// TwinCAT 3 PLC project State_Pattern
// Title: State Pattern PackML
// Company: ChrisK
// ProjectVersion: 0.0.0.1
// ProgramVersion: 3.1.4023.0
// libraries:
//   Tc2_Standard, * (Beckhoff Automation GmbH)
//   Tc2_System, * (Beckhoff Automation GmbH)
//   Tc3_Module, * (Beckhoff Automation GmbH)
//   Tc3_PackML_V2, * (Beckhoff Automation GmbH)
// project tree:
//   PackML_Method_Pattern/ PML_Method_Base.TcPOU
//   PackML_State_Pattern/ Aborted_State.TcPOU, Aborting_State.TcPOU, Clearing_State.TcPOU, Execute_State.TcPOU, Idle_State.TcPOU, ITF_State.TcIO, PML_StatePattern_Base.TcPOU, Resetting_State.TcPOU, Starting_State.TcPOU, Stopped_State.TcPOU, Undefined_State.TcPOU

// ---- PackML_State_Pattern/ITF_State.TcIO
INTERFACE ITF_State

METHOD Cycle : BOOL
VAR_INPUT
END_VAR
END_METHOD

END_INTERFACE

// ---- PackML_Method_Pattern/PML_Method_Base.TcPOU
FUNCTION_BLOCK PML_Method_Base
VAR_INPUT
END_VAR
VAR_OUTPUT
END_VAR
VAR
	ipackml : IPmlStateMachine;
END_VAR

METHOD PROTECTED Aborted : BOOL
VAR_INPUT
END_VAR
END_METHOD

METHOD PROTECTED Aborting : BOOL
VAR_INPUT
END_VAR
ipackml.SetStateComplete();
END_METHOD

METHOD PROTECTED Clearing : BOOL
VAR_INPUT
END_VAR
ipackml.SetStateComplete();
END_METHOD

METHOD PROTECTED Completed : BOOL
VAR_INPUT
END_VAR
END_METHOD

METHOD PROTECTED Completing : BOOL
VAR_INPUT
END_VAR
ipackml.SetStateComplete();
END_METHOD

METHOD PUBLIC Cycle : BOOL
VAR_INPUT
END_VAR
CASE ipackml.GetCurrentState() OF
	E_PMLState.ePMLState_Clearing:
		Clearing();
	E_PMLState.ePMLState_Aborted:
		Aborted();
	E_PMLState.ePMLState_Aborting:
		Aborting();
	E_PMLState.ePMLState_Complete:
		Completed();
	E_PMLState.ePMLState_Completing:
		Completing();
	E_PMLState.ePMLState_Execute:
		Execute();
	E_PMLState.ePMLState_Held:
		Held();
	E_PMLState.ePMLState_Holding:
		Holding();
	E_PMLState.ePMLState_Idle:
		Idle();
	E_PMLState.ePMLState_Resetting:
		Resetting();
	E_PMLState.ePMLState_Starting:
		Starting();
	E_PMLState.ePMLState_Stopped:
		Stopped();
	E_PMLState.ePMLState_Stopping:
		Stopping();
	E_PMLState.ePMLState_Suspended:
		Suspended();
	E_PMLState.ePMLState_Suspending:
		Suspending();
	E_PMLState.ePMLState_Undefined:
		Undefined();
	E_PMLState.ePMLState_Unholding:
		Unholding();
	E_PMLState.ePMLState_Unsuspending:
		Unsuspending();
END_CASE
END_METHOD

METHOD PROTECTED Execute : BOOL
VAR_INPUT
END_VAR
END_METHOD

METHOD PROTECTED Held : BOOL
VAR_INPUT
END_VAR
END_METHOD

METHOD PROTECTED Holding : BOOL
VAR_INPUT
END_VAR
ipackml.SetStateComplete();
END_METHOD

METHOD PROTECTED Idle : BOOL
VAR_INPUT
END_VAR
END_METHOD

PROPERTY PUBLIC PackMLStateMachine : IPmlStateMachine
GET
PackMLStateMachine := ipackml;
END_GET
SET
ipackml := PackMLStateMachine;
END_SET
END_PROPERTY

METHOD PROTECTED Resetting : BOOL
VAR_INPUT
END_VAR
ipackml.SetStateComplete();
END_METHOD

METHOD PROTECTED Starting : BOOL
VAR_INPUT
END_VAR
ipackml.SetStateComplete();
END_METHOD

METHOD PROTECTED Stopped : BOOL
VAR_INPUT
END_VAR
END_METHOD

METHOD PROTECTED Stopping : BOOL
VAR_INPUT
END_VAR
ipackml.SetStateComplete();
END_METHOD

METHOD PROTECTED Suspended : BOOL
VAR_INPUT
END_VAR
END_METHOD

METHOD PROTECTED Suspending : BOOL
VAR_INPUT
END_VAR
ipackml.SetStateComplete();
END_METHOD

METHOD PROTECTED Undefined : BOOL
VAR_INPUT
END_VAR
END_METHOD

METHOD PROTECTED Unholding : BOOL
VAR_INPUT
END_VAR
ipackml.SetStateComplete();
END_METHOD

METHOD PROTECTED Unsuspending : BOOL
VAR_INPUT
END_VAR
ipackml.SetStateComplete();
END_METHOD

END_FUNCTION_BLOCK

// ---- PackML_State_Pattern/Aborted_State.TcPOU
FUNCTION_BLOCK Aborted_State IMPLEMENTS ITF_State
VAR_INPUT
END_VAR
VAR_OUTPUT
END_VAR
VAR
	pPML_Base : POINTER TO PML_StatePattern_Base;
	_stateMachine : IPmlStateMachine;
END_VAR

METHOD Cycle : BOOL
VAR_INPUT
END_VAR
IF _stateMachine.GetCurrentState() = E_PMLState.ePMLState_Clearing THEN
	pPML_Base^.SetState(pPML_Base^.clearing);
END_IF
END_METHOD

METHOD FB_init : BOOL
VAR_INPUT
	bInitRetains : BOOL; // if TRUE, the retain variables are initialized (warm start / cold start)
	bInCopyCode : BOOL;  // if TRUE, the instance afterwards gets moved into the copy code (online change)
	pPML_Base : POINTER TO PML_StatePattern_Base;
	statemachine : IPmlStateMachine;
END_VAR
_stateMachine := statemachine;
THIS^.pPML_Base := pPML_Base;
END_METHOD

END_FUNCTION_BLOCK

// ---- PackML_State_Pattern/PML_StatePattern_Base.TcPOU
FUNCTION_BLOCK PML_StatePattern_Base
VAR_INPUT
END_VAR
VAR_OUTPUT
END_VAR
VAR
	stateMachine : PMLStateMachine;
	iStateMachine : IPmlStateMachine := stateMachine;
	undefined : Undefined_State(THIS, iStateMachine);
	aborting : Aborting_State(THIS, iStateMachine);
	aborted : Aborted_State(THIS, iStateMachine);
	clearing : Clearing_State(THIS, iStateMachine);
	stopped : Stopped_State(THIS, iStateMachine);
	resetting : Resetting_State(THIS, iStateMachine);
	idle : Idle_State(THIS, iStateMachine);
	starting : Starting_State(THIS, iStateMachine);
	execute : Execute_State(THIS, iStateMachine);
	iState : ITF_State := undefined;
END_VAR

iState.Cycle();
stateMachine();

METHOD SetState : BOOL
VAR_INPUT
  newState : ITF_State;
END_VAR
THIS^.iState := newState;
END_METHOD

END_FUNCTION_BLOCK

// ---- PackML_State_Pattern/Undefined_State.TcPOU
FUNCTION_BLOCK Undefined_State IMPLEMENTS ITF_State
VAR_INPUT
END_VAR
VAR_OUTPUT
END_VAR
VAR
	pPML_Base : POINTER TO PML_StatePattern_Base;
	_stateMachine : IPmlStateMachine;
END_VAR

METHOD Cycle : BOOL
VAR_INPUT
END_VAR
IF _stateMachine.GetCurrentState() = E_PMLState.ePMLState_Aborting THEN
	pPML_Base^.SetState(pPML_Base^.aborting);
END_IF
END_METHOD

METHOD FB_init : BOOL
VAR_INPUT
	bInitRetains : BOOL; // if TRUE, the retain variables are initialized (warm start / cold start)
	bInCopyCode : BOOL;  // if TRUE, the instance afterwards gets moved into the copy code (online change)
	pPML_Base : POINTER TO PML_StatePattern_Base;
	statemachine : IPmlStateMachine;
END_VAR
_stateMachine := statemachine;
THIS^.pPML_Base := pPML_Base;
END_METHOD

END_FUNCTION_BLOCK

// ---- PackML_State_Pattern/Aborting_State.TcPOU
FUNCTION_BLOCK Aborting_State  IMPLEMENTS ITF_State
VAR_INPUT
END_VAR
VAR_OUTPUT
END_VAR
VAR
	pPML_Base : POINTER TO PML_StatePattern_Base;
	_stateMachine : IPmlStateMachine;
END_VAR

METHOD Cycle : BOOL
_stateMachine.SetStateComplete();
pPML_Base^.SetState(pPML_Base^.aborted);
END_METHOD

METHOD FB_init : BOOL
VAR_INPUT
	bInitRetains : BOOL; // if TRUE, the retain variables are initialized (warm start / cold start)
	bInCopyCode : BOOL;  // if TRUE, the instance afterwards gets moved into the copy code (online change)
	pPML_Base : POINTER TO PML_StatePattern_Base;
	statemachine : IPmlStateMachine;
END_VAR
_stateMachine := statemachine;
THIS^.pPML_Base := pPML_Base;
END_METHOD

END_FUNCTION_BLOCK

// ---- PackML_State_Pattern/Clearing_State.TcPOU
FUNCTION_BLOCK Clearing_State  IMPLEMENTS ITF_State
VAR_INPUT
END_VAR
VAR_OUTPUT
END_VAR
VAR
	pPML_Base : POINTER TO PML_StatePattern_Base;
	_stateMachine : IPmlStateMachine;
END_VAR

METHOD Cycle : BOOL
_stateMachine.SetStateComplete();
pPML_Base^.SetState(pPML_Base^.stopped);
END_METHOD

METHOD FB_init : BOOL
VAR_INPUT
	bInitRetains : BOOL; // if TRUE, the retain variables are initialized (warm start / cold start)
	bInCopyCode : BOOL;  // if TRUE, the instance afterwards gets moved into the copy code (online change)
	pPML_Base : POINTER TO PML_StatePattern_Base;
	statemachine : IPmlStateMachine;
END_VAR
_stateMachine := statemachine;
THIS^.pPML_Base := pPML_Base;
END_METHOD

END_FUNCTION_BLOCK

// ---- PackML_State_Pattern/Stopped_State.TcPOU
FUNCTION_BLOCK Stopped_State  IMPLEMENTS ITF_State
VAR_INPUT
END_VAR
VAR_OUTPUT
END_VAR
VAR
	pPML_Base : POINTER TO PML_StatePattern_Base;
	_stateMachine : IPmlStateMachine;
END_VAR

METHOD Cycle : BOOL
VAR_INPUT
END_VAR
IF _stateMachine.GetCurrentState() = E_PMLState.ePMLState_Resetting THEN 
	pPML_Base^.SetState(pPML_Base^.resetting);
END_IF
END_METHOD

METHOD FB_init : BOOL
VAR_INPUT
	bInitRetains : BOOL; // if TRUE, the retain variables are initialized (warm start / cold start)
	bInCopyCode : BOOL;  // if TRUE, the instance afterwards gets moved into the copy code (online change)
	pPML_Base : POINTER TO PML_StatePattern_Base;
	statemachine : IPmlStateMachine;
END_VAR
_stateMachine := statemachine;
THIS^.pPML_Base := pPML_Base;
END_METHOD

END_FUNCTION_BLOCK

// ---- PackML_State_Pattern/Resetting_State.TcPOU
FUNCTION_BLOCK Resetting_State  IMPLEMENTS ITF_State
VAR_INPUT
END_VAR
VAR_OUTPUT
END_VAR
VAR
	pPML_Base : POINTER TO PML_StatePattern_Base;
	_stateMachine : IPmlStateMachine;
END_VAR

METHOD Cycle : BOOL
VAR_INPUT
END_VAR
_stateMachine.SetStateComplete();
pPML_Base^.SetState(pPML_Base^.idle);
END_METHOD

METHOD FB_init : BOOL
VAR_INPUT
	bInitRetains : BOOL; // if TRUE, the retain variables are initialized (warm start / cold start)
	bInCopyCode : BOOL;  // if TRUE, the instance afterwards gets moved into the copy code (online change)
	pPML_Base : POINTER TO PML_StatePattern_Base;
	statemachine : IPmlStateMachine;
END_VAR
_stateMachine := statemachine;
THIS^.pPML_Base := pPML_Base;
END_METHOD

END_FUNCTION_BLOCK

// ---- PackML_State_Pattern/Idle_State.TcPOU
FUNCTION_BLOCK Idle_State  IMPLEMENTS ITF_State
VAR_INPUT
END_VAR
VAR_OUTPUT
END_VAR
VAR
	pPML_Base : POINTER TO PML_StatePattern_Base;
	_stateMachine : IPmlStateMachine;
END_VAR

METHOD Cycle : BOOL
VAR_INPUT
END_VAR
IF _stateMachine.GetCurrentState() = E_PMLState.ePMLState_Starting THEN
	pPML_Base^.SetState(pPML_Base^.starting);
END_IF
END_METHOD

METHOD FB_init : BOOL
VAR_INPUT
	bInitRetains : BOOL; // if TRUE, the retain variables are initialized (warm start / cold start)
	bInCopyCode : BOOL;  // if TRUE, the instance afterwards gets moved into the copy code (online change)
	pPML_Base : POINTER TO PML_StatePattern_Base;
	statemachine : IPmlStateMachine;
END_VAR
_stateMachine := statemachine;
THIS^.pPML_Base := pPML_Base;
END_METHOD

END_FUNCTION_BLOCK

// ---- PackML_State_Pattern/Starting_State.TcPOU
FUNCTION_BLOCK Starting_State  IMPLEMENTS ITF_State
VAR_INPUT
END_VAR
VAR_OUTPUT
END_VAR
VAR
	pPML_Base : POINTER TO PML_StatePattern_Base;
	_stateMachine : IPmlStateMachine;
END_VAR

METHOD Cycle : BOOL
VAR_INPUT
END_VAR
_stateMachine.SetStateComplete();
pPML_Base^.SetState(pPML_Base^.execute);
END_METHOD

METHOD FB_init : BOOL
VAR_INPUT
	bInitRetains : BOOL; // if TRUE, the retain variables are initialized (warm start / cold start)
	bInCopyCode : BOOL;  // if TRUE, the instance afterwards gets moved into the copy code (online change)
	pPML_Base : POINTER TO PML_StatePattern_Base;
	statemachine : IPmlStateMachine;
END_VAR
_stateMachine := statemachine;
THIS^.pPML_Base := pPML_Base;
END_METHOD

END_FUNCTION_BLOCK

// ---- PackML_State_Pattern/Execute_State.TcPOU
FUNCTION_BLOCK Execute_State  IMPLEMENTS ITF_State
VAR_INPUT
END_VAR
VAR_OUTPUT
END_VAR
VAR
	pPML_Base : POINTER TO PML_StatePattern_Base;
	_stateMachine : IPmlStateMachine;
END_VAR

METHOD Cycle : BOOL
VAR_INPUT
END_VAR
IF _stateMachine.GetCurrentState() = E_PMLState.ePMLState_Aborting THEN
	pPML_Base^.SetState(pPML_Base^.aborting);
END_IF
END_METHOD

METHOD FB_init : BOOL
VAR_INPUT
	bInitRetains : BOOL; // if TRUE, the retain variables are initialized (warm start / cold start)
	bInCopyCode : BOOL;  // if TRUE, the instance afterwards gets moved into the copy code (online change)
	pPML_Base : POINTER TO PML_StatePattern_Base;
	statemachine : IPmlStateMachine;
END_VAR
_stateMachine := statemachine;
THIS^.pPML_Base := pPML_Base;
END_METHOD

END_FUNCTION_BLOCK
